Universal Robots PolyScope program: move_path_3right.urp

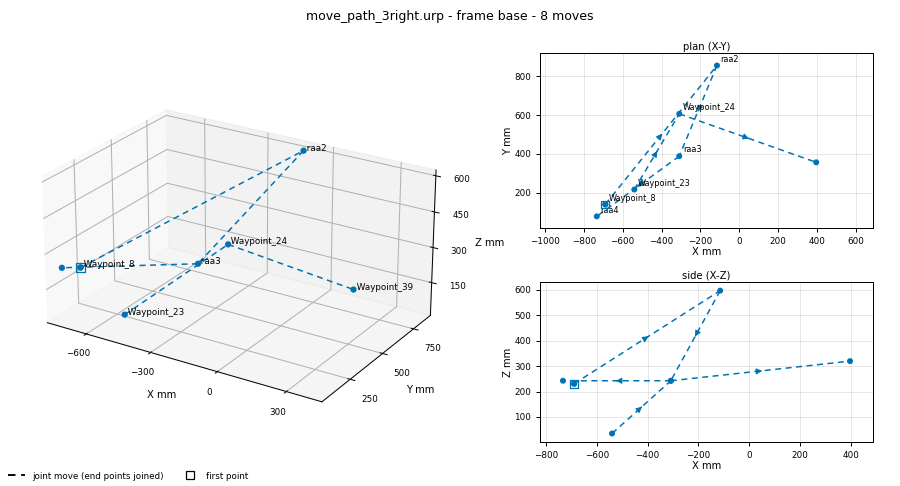
[picture p0: tool path of move_path_3right.urp in frame base, 8 of 23 moves have a stored position in this frame; points joined in program order, loops and branches not executed]
Program move_path_3right_1 (installation=default directory=/programs createdIn=5.21.3 lastSavedIn=5.21.3 robotSerialNumber=20246801938)
Calibrated DH parameters: a=[-0.000071, -0.790281, -0.600694, 0.000061, -0.000039, 0]; d=[0.236272, 604.465945, 132.116513, -736.382239, 0.159268, 0.154005]; alpha=[1.570254, -0.000567, 0.000559, 1.571709, -1.56999, 0]; deltaTheta=[0, -0.409357, 7.293326, -0.600784, -0.000001, -0.000001]
InitVariablesNode variables(variable(name=free_dr_already, expression=False), variable(name=freedrive_m_var, expression=False))
Robot Program (runOnlyOnce=false)
  'this is the path for Down, Over, then Back Around'
  ''
  SuppressedNode
    MoveJ speed 60 deg/s, acceleration 80 deg/s^2 (useActiveTCP=true optimoveEnabled=false optiMoveSpeed=0.3 optiMoveAcceleration=0.09) feature=Base
      Waypoint Waypoint_6: TCP in base x=-184.857 y=475.908 z=794.864 mm, rx=-0.225 ry=-1.9295 rz=0.6849 rad; joints [-137.383, -87.857, 120.236, 55.281, -50.736, -25.25] deg; TCP offset x=-5.053 y=-331.71 z=103.574 mm, rx=1.2092 ry=-1.2092 rz=1.2092 rad
      Waypoint Waypoint_1: TCP in base x=-161.037 y=970.524 z=722.042 mm, rx=-0.555 ry=0.1065 rz=0.3286 rad; joints [-74.895, -76.586, 126.53, 213.07, -169.134, 52.325] deg; TCP offset x=-4.211 y=-279.829 z=105.916 mm, rx=1.2092 ry=-1.2092 rz=1.2092 rad
      Waypoint Waypoint_7: TCP in base x=-689.651 y=138.963 z=230.691 mm, rx=-0.852 ry=-1.646 rz=1.646 rad; joints [-53.938, -86.03, 160.535, 285.425, -269.23, 90.049] deg
      SuppressedNode
        Waypoint Waypoint_1: TCP in base x=-1177.596 y=138.956 z=230.69 mm, rx=-0.852 ry=-1.646 rz=1.646 rad; joints [-20.637, -63.427, 120.718, 302.664, -235.94, 90.036] deg
      SuppressedNode
        Waypoint Waypoint_2: TCP in base x=-689.651 y=138.963 z=230.691 mm, rx=-0.852 ry=-1.646 rz=1.646 rad; joints [-53.938, -86.03, 160.535, 285.425, -269.23, 90.049] deg
      SuppressedNode
        Waypoint Waypoint_3: TCP in base x=-161.037 y=970.524 z=722.042 mm, rx=-0.555 ry=0.1065 rz=0.3286 rad; joints [-74.895, -76.586, 126.53, 213.07, -169.134, 52.325] deg
      SuppressedNode
        SafeHome (positionOptionType=SPEED_AND_ACCELERATION speed=1.047198 acceleration=1.396263 nextMotionTime=2)
  Script: align_ready_for_welding()
  ''
  p1 := pathturn[0]
  p2 := pathturn[1]
  p4 := pathturn[2]
  p5 := pathturn[3]
  pa1 := p[p1[0]+0.05,p1[1]+0.05,p1[2],p1[3],p1[4],p1[5]]
  liftcolumnz := liftcolumnzneeded
  URCap MachineLogic for Universal Robots (MachineLogic for Universal Robots, Vention Inc.) dataModel(type=addMotor, numberAdded=0, speed_in_mm_per_min=600, acceleration_in_mm_per_s2=50.0, ActuatorPos=liftcolumnz, teachColor=BLUE, combo1=MachineMotion1, combo2=(1) Custom Actuator, combo3=Move to Position, combo6=In series, message=Move to Position, description=Moves the actuator to a specified position from the home location., comboAddress=Address 1, comboActuator=Valve 1)
  MoveJ speed 20 deg/s, acceleration 80 deg/s^2 (useActiveTCP=true optimoveEnabled=false optiMoveSpeed=0.3 optiMoveAcceleration=0.09) feature=Base
    Waypoint Variable (Variable): variable=pa1
  MoveL speed 50 mm/s, acceleration 200 mm/s^2 (useActiveTCP=true optimoveEnabled=false optiMoveSpeed=0.3 optiMoveAcceleration=0.09) feature=Base
    Waypoint Variable (Variable): variable=p1
  Wait Sleep waitTime=8
  URCap WireTank Serial (WireTank Serial, WireTank, LLC) dataModel(NODE_TITLE=Serial Bridge uR1, Command=[252,82,49], QUERY=false, OUTPUT_ENTRY=Static, byte_array=true, Variable(key=OUTPUT_VARIABLE, variable(name=HwResp)))
  URCap WireTank Serial (WireTank Serial, WireTank, LLC) dataModel(NODE_TITLE=Serial Bridge uR1, Command=[252,82,49], QUERY=false, byte_array=true, OUTPUT_ENTRY=Static, Variable(key=OUTPUT_VARIABLE, variable(name=HwResp)))
  Wait Sleep waitTime=1
  SuppressedNode
    Script: turn_extrusion_on()
  Set DigitalOutput pin=digital_out[0]; digitalValue=1
  MoveL speed 10 mm/s, acceleration 100 mm/s^2 (useActiveTCP=true optimoveEnabled=false optiMoveSpeed=0.3 optiMoveAcceleration=0.09) feature=Base
    Waypoint Variable (Variable): variable=p2
  URCap WireTank Serial (WireTank Serial, WireTank, LLC) dataModel(QUERY=false, NODE_TITLE=Serial Bridge uR0, Command=[252,82,48], OUTPUT_ENTRY=Static, byte_array=true, Variable(key=OUTPUT_VARIABLE, variable=HwResp))
  Wait Sleep waitTime=0.5
  Set DigitalOutput pin=digital_out[0]; digitalValue=0
  MoveL speed 120 mm/s, acceleration 10 mm/s^2 (useActiveTCP=true optimoveEnabled=false optiMoveSpeed=0.3 optiMoveAcceleration=0.09) feature=Base
    Waypoint Variable (Variable): variable=p4
  URCap WireTank Serial (WireTank Serial, WireTank, LLC) dataModel(NODE_TITLE=Serial Bridge uR1, Command=[252,82,49], QUERY=false, byte_array=true, OUTPUT_ENTRY=Static, Variable(key=OUTPUT_VARIABLE, variable=HwResp))
  URCap WireTank Serial (WireTank Serial, WireTank, LLC) dataModel(NODE_TITLE=Serial Bridge uR1, Command=[252,82,49], byte_array=true, OUTPUT_ENTRY=Static, QUERY=false, Variable(key=OUTPUT_VARIABLE, variable=HwResp))
  Wait Sleep waitTime=1
  SuppressedNode
    Script: turn_extrusion_on()
  Set DigitalOutput pin=digital_out[0]; digitalValue=1
  MoveL speed 10 mm/s, acceleration 100 mm/s^2 (useActiveTCP=true optimoveEnabled=false optiMoveSpeed=0.3 optiMoveAcceleration=0.09) feature=Base
    Waypoint Variable (Variable): variable=p5
  URCap WireTank Serial (WireTank Serial, WireTank, LLC) dataModel(QUERY=false, NODE_TITLE=Serial Bridge uR0, Command=[252,82,48], byte_array=true, OUTPUT_ENTRY=Static, Variable(key=OUTPUT_VARIABLE, variable=HwResp))
  Wait Sleep waitTime=2
  Set DigitalOutput pin=digital_out[0]; digitalValue=0
  ''
  pret1 := p[p5[0]+.1,p5[1],p5[2],p5[3],p5[4],p5[5]]
  p_1 := pathturn[4]
  p_2 := pathturn[5]
  p_3 := pathturn[6]
  p_4 := pathturn[7]
  p_5 := pathturn[8]
  p_preheat := p[p_3[0]+.01,p_3[1],p_3[2],p_3[3],p_3[4],p_3[5]]
  p_pre_ret := p[p_1[0]+.03,p_1[1]+.03,p_1[2],p_1[3],p_1[4],p_1[5]]
  p_pre_ret2 := p[p_3[0]+.1,p_3[1],p_3[2],p_3[3],p_3[4],p_3[5]]
  'twist'
  MoveJ speed 80 deg/s, acceleration 80 deg/s^2 (useActiveTCP=true optimoveEnabled=false optiMoveSpeed=0.3 optiMoveAcceleration=0.09) feature=Base
    Waypoint Variable (Variable): variable=pret1
    Waypoint Waypoint_8: motionParameters(jointSpeed=1.047198 jointAcceleration=1.396263 cartesianSpeed=0.25 cartesianAcceleration=1.2); TCP in base x=-689.651 y=138.963 z=230.691 mm, rx=-0.852 ry=-1.646 rz=1.646 rad; joints [-53.938, -86.03, 160.535, 285.425, -269.23, 90.049] deg
    SuppressedNode
      Waypoint Waypoint_22: TCP in base x=-308.534 y=606.085 z=242.393 mm, rx=1.3699 ry=1.0669 rz=-1.2572 rad; joints [-84.142, -55.374, 92.791, 53.186, 94.965, 15.074] deg
  MoveJ speed 60 deg/s, acceleration 80 deg/s^2 (useActiveTCP=true optimoveEnabled=false optiMoveSpeed=0.3 optiMoveAcceleration=0.09) feature=Base
    Waypoint raa1: TCP in base x=-689.643 y=139.074 z=230.691 mm, rx=-0.8521 ry=-1.6459 rz=1.6459 rad; joints [-65.636, -88.39, 163.033, 285.277, -280.919, 90.061] deg; TCP offset x=-5.49 y=-328 z=106.39 mm, rx=1.2092 ry=-1.2092 rz=1.2092 rad
    Waypoint raa2: TCP in base x=-114.157 y=855.108 z=597.477 mm, rx=-0.5059 ry=0.3258 rz=0.3887 rad; joints [-71.965, -76.72, 138.376, 209.36, -156.862, 65.09] deg
    Waypoint raa3: TCP in base x=-308.547 y=387.798 z=242.407 mm, rx=1.9763 ry=0.3502 rz=-1.916 rad; joints [-108.471, -75.035, 126.793, 41.355, 93.912, 46.558] deg
    Waypoint raa4: TCP in base x=-733.576 y=77.691 z=242.41 mm, rx=1.9764 ry=0.3501 rz=-1.9161 rad; joints [-51.046, -76.954, 130.276, 41.633, 89.45, 103.864] deg
    SuppressedNode
      Waypoint Waypoint_2: TCP in base x=-308.546 y=606.076 z=242.404 mm, rx=1.3699 ry=1.0669 rz=-1.2572 rad; joints [-84.814, -53.028, 88.323, 55.251, 94.969, 14.398] deg
  If liftcolumnz≠0.0
    URCap MachineLogic for Universal Robots (MachineLogic for Universal Robots, Vention Inc.) dataModel(type=addMotor, numberAdded=0, speed_in_mm_per_min=600, acceleration_in_mm_per_s2=50.0, teachColor=BLUE, combo1=MachineMotion1, combo2=(1) Custom Actuator, combo3=Home, combo6=In series, message=Homing, description=Moves the actuator in the negative direction until the home sensor is triggered and sets position to zero (0)., comboAddress=Address 1, comboActuator=Valve 1)
  'preheat'
  SuppressedNode
    MoveJ speed 60 deg/s, acceleration 80 deg/s^2 (useActiveTCP=true optimoveEnabled=false optiMoveSpeed=0.3 optiMoveAcceleration=0.09) feature=Base
      Waypoint Variable (Variable): variable=p_pre_ret
  MoveL speed 250 mm/s, acceleration 1200 mm/s^2 (useActiveTCP=true optimoveEnabled=false optiMoveSpeed=0.3 optiMoveAcceleration=0.09) feature=Base
    Waypoint Variable (Variable): variable=p_pre_ret2
    Waypoint Variable (Variable): variable=p_preheat
  Wait Sleep waitTime=6
  MoveL speed 250 mm/s, acceleration 1200 mm/s^2 (useActiveTCP=true optimoveEnabled=false optiMoveSpeed=0.3 optiMoveAcceleration=0.09) feature=Base
    Waypoint Variable (Variable): variable=p_pre_ret2
    Waypoint Variable (Variable): variable=p_pre_ret
  Set NoAction tcp=backofhole
  MoveL speed 50 mm/s, acceleration 1200 mm/s^2 (useActiveTCP=true optimoveEnabled=false optiMoveSpeed=0.3 optiMoveAcceleration=0.09) feature=Base
    Waypoint Variable (Variable): variable=p_1
  URCap WireTank Serial (WireTank Serial, WireTank, LLC) dataModel(NODE_TITLE=Serial Bridge uR1, Command=[252,82,49], QUERY=false, byte_array=true, OUTPUT_ENTRY=Static, Variable(key=OUTPUT_VARIABLE, variable=HwResp))
  URCap WireTank Serial (WireTank Serial, WireTank, LLC) dataModel(NODE_TITLE=Serial Bridge uR1, Command=[252,82,49], QUERY=false, byte_array=true, OUTPUT_ENTRY=Static, Variable(key=OUTPUT_VARIABLE, variable=HwResp))
  Wait Sleep waitTime=1
  Set DigitalOutput pin=digital_out[0]; digitalValue=1
  SuppressedNode
    Script: turn_extrusion_on()
  Wait Sleep waitTime=1
  MoveL speed 10 mm/s, acceleration 1200 mm/s^2 (useActiveTCP=true optimoveEnabled=false optiMoveSpeed=0.3 optiMoveAcceleration=0.09) feature=Base
    Waypoint Variable (Variable): variable=p_2
  MoveP speed 0.5 mm/s, acceleration 10 mm/s^2 (blendRadius=0.001 useActiveTCP=true optimoveEnabled=false optiMoveSpeed=0.3 optiMoveAcceleration=0.09) feature=Base
    CircleMove (OrientationMode=FIXED)
      Waypoint Variable (Variable): variable=p_3
      Waypoint Variable (Variable): variable=p_4
  MoveL speed 12 mm/s, acceleration 1200 mm/s^2 (useActiveTCP=true optimoveEnabled=false optiMoveSpeed=0.3 optiMoveAcceleration=0.09) feature=Base
    Waypoint Variable (Variable): variable=p_5
  URCap WireTank Serial (WireTank Serial, WireTank, LLC) dataModel(QUERY=false, NODE_TITLE=Serial Bridge uR0, Command=[252,82,48], OUTPUT_ENTRY=Static, byte_array=true, Variable(key=OUTPUT_VARIABLE, variable=HwResp))
  Wait Sleep waitTime=2
  Set DigitalOutput pin=digital_out[0]; digitalValue=0
  MoveL speed 250 mm/s, acceleration 1200 mm/s^2 (useActiveTCP=true optimoveEnabled=false optiMoveSpeed=0.3 optiMoveAcceleration=0.09) feature=Base
    Waypoint Waypoint_23: TCP in base x=-540.167 y=215.949 z=34.631 mm, rx=-1.5058 ry=1.0576 rz=1.5735 rad; joints [-26.452, -65.119, 143.749, 8.723, 85.674, 218.843] deg; TCP offset x=-4.211 y=-279.829 z=105.916 mm, rx=1.2092 ry=-1.2092 rz=1.2092 rad
  MoveJ speed 60 deg/s, acceleration 80 deg/s^2 (useActiveTCP=true optimoveEnabled=false optiMoveSpeed=0.3 optiMoveAcceleration=0.09) feature=Base
    Waypoint Waypoint_24: TCP in base x=-308.526 y=606.096 z=242.373 mm, rx=-2.1337 ry=0.3494 rz=2.1309 rad; joints [-107.196, -73.784, 125.643, 43.029, 90.975, 86.468] deg
    Waypoint Waypoint_39: TCP in base x=397.377 y=356.253 z=319.81 mm, rx=2.3163 ry=2.0576 rz=0.0741 rad; joints [-198.126, -117.851, 133.304, -13.01, -11.422, -6.036] deg; TCP offset x=-5.49 y=-328 z=106.39 mm, rx=1.2092 ry=-1.2092 rz=1.2092 rad
    'above waypoint is home'
